// TIA Portal V16 export
// export: Created 2021-07-12T14:47:20.0834697Z, ExportSetting WithDefaults, DisplayName Totally Integrated Automation Portal, DisplayVersion V16, DisplayName TIA Portal Version Control Interface, DisplayVersion V16, DisplayName TIA Portal Openness, DisplayVersion V16, DisplayName STEP 7 Professional, DisplayVersion V16, DisplayName STEP 7 Safety, DisplayVersion V16, DisplayName WinCC Professional, DisplayVersion V16
TYPE "SimaHydTO_typeHMIConnectionBasicAxisControlCommand"
TITLE = SimaHydTO_typeHMIConnectionBasicAxisControlCommand
// HMI interface: Basic axis control (LAxisBasics) - Command (HMI -> PLC)
// stored: IsFailsafeCompliant false
   STRUCT
      powerEnable : Bool;   // MC_Power: 0: The technology object is disabled / 1: The technology object is enabled
      powerStartMode : DInt := 1;   // 0: Enable axis not position-controlled / 1: Enable axis position-controlled
      powerStopMode : Int := 0;   // 0: Emergency stop / 1: Immediate stop / 2: Stop with maximum dynamic values
      resetExecute : Bool;   // MC_Reset: Start job with a positive edge
      resetFBExecute : Bool;   // LSimaHyd_MC_Reset: Start job with a positive edge
      resetRestart : Bool := false;   // 0: Acknowledgment of queued technology alarms / 1: Reinitialization of the technology object and acknowledgment of pending technology alarms
      homeExecute : Bool;   // MC_Home: Start job with a positive edge
      homePosition : LReal;   // The specified value is used according to the selected "Mode".
      homeMode : Int;   // 0: Direct homing (absolute) / 1: Direct homing (relative) / 2: Passive homing / 3: Active homing / 4: Reserved / 5: Active homing (<TO>.Homing.HomePosition) / 6: Absolute encoder adjustment (relative) / 7: Absolute encoder adjustment (absolute) / 8: Passive homing / 9: Abort passive homing / 10: Passive homing (<TO>.Homing.HomePosition)
      jogForward : Bool;   // MC_MoveJog: As long as the parameter is TRUE, the axis moves in the positive direction
      jogBackward : Bool;   // MC_MoveJog: As long as the parameter is TRUE, the axis moves in the negative direction
      jogVelocity : LReal := 100.0;   // Velocity setpoint / speed setpoint for the motion
      jogAcceleration : LReal := -1.0;   // Acceleration of jog movement
      jogDeceleration : LReal := -1.0;   // Deceleration of jog movement
      jogJerk : LReal := -1.0;   // Jerk of jog movement
      jogPositionControlled : Bool := true;   // 0: Non position-controlled operation / 1: Position-controlled mode - The parameter applies as long as the MC_MoveJog command is executed. After this, the setting of MC_Power applies again.
   END_STRUCT;
END_TYPE
